FUNCTION_BLOCK FB_FCSLBaseKeyValueLogMsgListener EXTENDS FB_ListenerBase2
VAR
    json          			: FB_JsonDomParser; 		//Parse JSON attribute of messages
    jsonAttribute 			: STRING(10000);    		//Holds JSON attribute
    hr           			: HRESULT;         		//Signals JSON attribute was successfully read
    ipListener    			: I_KeyValueLogListener; 	//Receives callback once message is processed
	
	fbRequestEventText 		: FB_RequestEventText;
	{attribute 'TcEncoding':='UTF-8'}
	sLastMessageText 		: STRING;
	
END_VAR

PROPERTY Listener : I_KeyValueLogListener
SET
ipListener := Listener;
END_SET
END_PROPERTY

METHOD OnMessageSent : Tc3_EventLogger.HRESULT
VAR_INPUT
    fbEvent 			: REFERENCE TO FB_TcEvent;
END_VAR

VAR
    message      		: ST_KeyValueLogMessages;
    jsonDocument 		: SJsonValue;
    jsonProperty 		: SJsonValue;
	jsonExtendedInfo	: SJsonValue;
	
	bHasMember 			: BOOL;
END_VAR
hr := fbEvent.GetJsonAttribute(JsonAttribute, SIZEOF(JsonAttribute));

IF ( SUCCEEDED(hr) ) THEN
    jsonDocument := json.ParseDocument(jsonAttribute);

    IF ( json.HasMember(jsonDocument, 'Timestamp') ) THEN
        jsonProperty      := json.FindMember(jsonDocument, 'Timestamp');
        message.Timestamp := json.GetString(jsonProperty);
    END_IF

    IF ( json.HasMember(jsonDocument, 'k') ) THEN
        jsonProperty    := json.FindMember(jsonDocument, 'k');
        message.k := json.GetString(jsonProperty);
    END_IF
	
    IF ( json.HasMember(jsonDocument, 'v') ) THEN
        jsonProperty    := json.FindMember(jsonDocument, 'v');
 		message.v := json.GetString(jsonProperty);
    END_IF

    IF ( ipListener <> 0 ) THEN
        //Notify listener of message data
        ipListener.OnTraceReceived(Message);
    END_IF
END_IF

OnMessageSent := S_OK; // in order to receive more callbacks (Set <> S_OK in order to cancel the callbacks for this program cycle.)
END_METHOD

END_FUNCTION_BLOCK

(* stored: Version 1.1.0.1
   POU FB_FCSLBaseKeyValueLogMsgListener: Id {89058bac-53af-4255-8c0f-080af613db25}, SpecialFunc None
   Property Listener: Id {7495434e-7678-4692-8389-fa3f59c84f89}
   Set Set: Id {251fc7d5-2ccf-4c12-8e6d-7ed11ac5f367}
   Method OnMessageSent: Id {a1cb46a8-aede-4059-ab08-87fbece9f8d1} *)
